% RSLogix 500 project average.RSS, saved by version 8.30.00.15 %
PROJECT "UNTITLED"    % processor: MicroLogix 1000 %

PROGRAM FILES
  LAD 2 "MAIN_PROG"  2 rungs
  LAD 3 "USER_FAULT"  1 rungs
  LAD 4 "HSC_INT"  1 rungs
  LAD 5 "STI_INT"  1 rungs
  LAD 6, 7, 8, 9, 10, 11, 12, 13, 14, 15, 16: only END

DATA FILES
  O0 OUTPUT  1 elements
  I1 INPUT  2 elements
  S2 STATUS  33 elements
  B3 BINARY  32 elements
  T4 TIMER  40 elements
  C5 COUNTER  32 elements
  R6 CONTROL  16 elements
  N7 INTEGER  105 elements

LADDER 2 "MAIN_PROG"
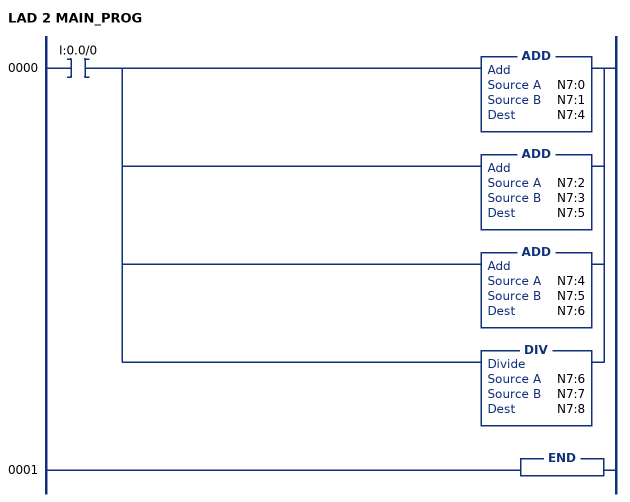
% Rung: 0 %
SOR XIC I:0.0/0 BST BST BST ADD N7:0 N7:1 N7:4 NXB ADD N7:2 N7:3 N7:5 BND NXB ADD N7:4 N7:5 N7:6 BND NXB DIV N7:6 N7:7 N7:8 BND EOR
% Rung: 1 %
SOR END EOR

DATA TABLE (non-zero values as saved)
DATA N7
% N7:0 % 4 8 6 10 12 16 28 4 7 0
